    end
    $ 1242 "MoveJ"
    $ 1243 "CaptPos0" "breakAfter"
    set_tcp(p[0.0,0.0,0.0,0.0,0.0,0.0])
    movej(get_inverse_kin(CaptPos0_p, qnear=CaptPos0_q), a=0.2617993877991494, v=0.15707963267948966)
  end
  def SUB_6101():
    $ 1244 "SUB_6101" "noBreak"
    $ 1245 "ROVI_RECIPE"
    $ 1246 "If文 (not ROVI_RECIPE(GPII_WorkNo))"
    if ((not ROVI_RECIPE(read_input_integer_register(2)))):
      $ 1247 "SubPrgResult:=rovi_err"
      global SubPrgResult=rovi_err
      $ 1248 "待機: 999999.0"
      sleep(999999.0)
    end
    $ 1249 "ROVI_RESET"
    $ 1250 "If文 ( not ROVI_RESET())"
    if ((  not  ROVI_RESET())):
      $ 1251 "SubPrgResult:=rovi_err"
      global SubPrgResult=rovi_err
      $ 1252 "待機: 999999.0"
      sleep(999999.0)
    end
    $ 1253 "ROVI_CAPTURE_1"
    $ 1254 "MoveJ"
    $ 1255 "スイッチ文 CheckMST"
    switch_1 = CheckMST
    $ 1256 "ケース 0"
    if (0 == switch_1):
      $ 1257 "Master_pos" "breakAfter"
      set_tcp(p[0.0,0.09,0.42,0.0,0.0,0.0])
      movej(Master_pos, a=0.20943951023931953, v=0.10471975511965977)
    elif (1 == switch_1):
      $ 1258 "ケース 1"
      $ 1259 "Master_pos" "breakAfter"
      set_tcp(p[0.0,0.09,0.42,0.0,0.0,0.0])
      movej(Master_pos, a=0.20943951023931953, v=0.10471975511965977)
    elif (2 == switch_1):
      $ 1260 "ケース 2"
      $ 1261 "Master_posL" "breakAfter"
      set_tcp(p[0.0,0.09,0.42,0.0,0.0,0.0])
      movej(Master_posL, a=0.20943951023931953, v=0.10471975511965977)
    elif (3 == switch_1):
      $ 1262 "ケース 3"
      $ 1263 "Master_posR" "breakAfter"
      set_tcp(p[0.0,0.09,0.42,0.0,0.0,0.0])
      movej(Master_posR, a=0.20943951023931953, v=0.10471975511965977)
    end
    $ 1265 "待機: 3.0"
    sleep(3.0)
    $ 1266 "If文 ( not ROVI_CAPTURE())"
    if ((  not  ROVI_CAPTURE())):
      $ 1267 "SubPrgResult:=rovi_err"
      global SubPrgResult=rovi_err
      $ 1268 "待機: 999999.0"
      sleep(999999.0)
    end
  end
  def SUB_6102RXFF():
    $ 1438 "SUB_6102RXFF" "noBreak"
    $ 1439 "荷重の設定: k10"
    set_target_payload(0.100000, [0.135000, 0.000000, 0.225000], [10.000000, 10.000000, 10.000000, 0.000000, 0.000000, 0.000000])
    $ 1440 "UF:=ベース_const"
    global UF=p[0.0,0.0,0.0,0.0,0.0,0.0]
    $ 1441 "If文 (GPII_CheckMST>0)"
    if ((read_input_integer_register(23)>0)):
      $ 1442 "ROVI_SOLVE"
      $ 1443 "If文 (CandCnt>0)"
      if ((CandCnt>0)):
        $ 1444 "Y2:=ROVI_SOLVE()"
        global Y2=ROVI_SOLVE()
        $ 1445 "If文 (Y2[0]≟10000.)"
        if ((Y2[0] == 10000.)):
          $ 1446 "SubPrgResult:=rovi_err"
          global SubPrgResult=rovi_err
          $ 1447 "待機: 999999.0"
          sleep(999999.0)
        end
      end
      $ 1448 "UF:=Y2"
      global UF=Y2
    end
    $ 1449 "M"
    $ 1450 "MoveL"
    $ 1451 "gGD_3_M_RX" "breakAfter"
    set_tcp(p[0.0,0.09,0.42,1.894,0.0,0.0])
    movel(pose_trans(UF, gGD_3_M_RX), a=0.07, v=0.12)
    $ 1452 "待機: 1.0"
    sleep(1.0)
    $ 1453 "gGD_2_M_RX" "breakAfter"
    set_tcp(p[0.0,0.09,0.42,1.894,0.0,0.0])
    movel(pose_trans(UF, gGD_2_M_RX), a=0.07, v=0.12)
    $ 1454 "待機: 1.0"
    sleep(1.0)
    $ 1455 "設定 GPBO_BLStop=HI:Pulse 1.0"
    thread SinglePulse2252():
      write_output_boolean_register(14, True)
      sleep(1.0)
      write_output_boolean_register(14, False)
    end
    singlePulse2252 = run SinglePulse2252()
    $ 1456 "ポップアップ: ok?"
    popup("ok?", "メッセージ", False, False, blocking=True)
    $ 1457 "tm_6102_01: リセット"
    tm_6102_01 = 0
    $ 1458 "tm_6102_01: 起動"
    tm_6102_01_is_counting = True
    $ 1459 "フォース"
    sleep(0.02)
    zero_ftsensor()
    force_mode(tool_pose(), [1, 1, 1, 0, 0, 0], [0.0, 0.0, 10.0, 0.0, 0.0, 0.0], 2, [0.005, 0.005, 0.04, 0.3490658503988659, 0.3490658503988659, 0.3490658503988659])
    $ 1460 "ShakeCnt:=-1" "noBreak"
    global ShakeCnt=-1
    $ 1461 "ループ ((Currpos_p_UF0[1]>(gGD_2_M_RX[1]-HandInZ)) and (tm_6102_01<GPII_TMHandIn))" "noBreak"
    while (((Currpos_p_UF0[1]>(gGD_2_M_RX[1]-HandInZ))  and  (tm_6102_01<read_input_integer_register(12)))):
      $ 1462 "IsShake:= False " "noBreak"
      global IsShake=  False
      $ 1463 "If文 ShakeCnt<0" "noBreak"
      if (ShakeCnt<0):
        $ 1464 "NOT_SHAKE" "noBreak"
        $ 1465 "tm_6102_02: 起動" "noBreak"
        tm_6102_02_is_counting = True
        $ 1466 "待機 tm_6102_02>ShakeWaitSec" "noBreak"
        while (not(tm_6102_02>ShakeWaitSec)):
          sync()
        end
        $ 1467 "tm_6102_02: 停止" "noBreak"
        tm_6102_02_is_counting = False
        $ 1468 "tm_6102_02: リセット" "noBreak"
        tm_6102_02 = 0
        $ 1469 "ShakeCnt:=0" "noBreak"
        global ShakeCnt=0
      end
      $ 1470 "MONITOR_SPEED" "noBreak"
      $ 1471 "tm_6102_02: リセット" "noBreak"
      tm_6102_02 = 0
      $ 1472 "If文 norm(TCPSpeed[2])<TCPSpeedThZ" "noBreak"
      if (norm(TCPSpeed[2])<TCPSpeedThZ):
        $ 1473 "IsShake:= True " "noBreak"
        global IsShake=  True
        $ 1474 "If文 ShakeCnt≟0" "noBreak"
        if (ShakeCnt == 0):
          $ 1475 "tm_6102_02: 起動" "noBreak"
          tm_6102_02_is_counting = True
          $ 1476 "ループ ((tm_6102_02<1.0) and (IsShake≟ True ))" "noBreak"
          while (((tm_6102_02<1.0)  and  (IsShake ==   True  ))):
            $ 1477 "If文 norm(TCPSpeed[2])≥TCPSpeedThZ" "noBreak"
            if (norm(TCPSpeed[2]) >= TCPSpeedThZ):
              $ 1478 "IsShake:= False " "noBreak"
              global IsShake=  False
            end
          end
          $ 1479 "tm_6102_02: 停止" "noBreak"
          tm_6102_02_is_counting = False
        end
        $ 1480 "ShakeCnt:=ShakeCnt+1" "noBreak"
        global ShakeCnt=ShakeCnt+1
      end
      $ 1481 "SHAKE" "noBreak"
      $ 1482 "If文 IsShake" "noBreak"
      if (IsShake):
        $ 1483 "Sub3100_Option:=9" "noBreak"
        global Sub3100_Option=9
        $ 1484 "ループ2回" "noBreak"
        u12523u12540u12503_6 = 0
        while (u12523u12540u12503_6 < 2):
          $ 1485 "'7:RX+,8:RX-,9:RY+,10:RY-,11:RZ+,12:RZ-'" "noBreak"
          # '7:RX+,8:RX-,9:RY+,10:RY-,11:RZ+,12:RZ-'
          $ 1486 "Sub3100_Xd:=[0.,0.,0.,0.,0.,0.]" "noBreak"
          global Sub3100_Xd=[0.,0.,0.,0.,0.,0.]
          $ 1487 "Sub3100_q:=floor((Sub3100_Option-1) / 2)" "noBreak"
          global Sub3100_q=floor((Sub3100_Option-1) / 2)
          $ 1488 "Sub3100_e:=1-((Sub3100_Option-1) % 2)*2" "noBreak"
          global Sub3100_e=1-((Sub3100_Option-1) % 2)*2
          $ 1489 "Sub3100_t:=0.2" "noBreak"
          global Sub3100_t=0.2
          $ 1490 "Sub3100_Xd[Sub3100_q]=d2r(Sub3100_XdRot/2.0)*Sub3100_e" "noBreak"
          Sub3100_Xd[Sub3100_q]= d2r (Sub3100_XdRot/2.0)*Sub3100_e
          $ 1491 "speedl(Sub3100_Xd,Sub3100_aRot/2.0,Sub3100_t)" "noBreak"
          speedl(Sub3100_Xd,Sub3100_aRot/2.0,Sub3100_t)
          $ 1492 "If文 Sub3100_Option≟9" "noBreak"
          if (Sub3100_Option == 9):
            $ 1493 "Sub3100_Option:=10" "noBreak"
            global Sub3100_Option=10
          else:
            $ 1494 "Else" "noBreak"
            $ 1495 "Sub3100_Option:=9" "noBreak"
            global Sub3100_Option=9
          end
          $ 1496 "待機: 0.1" "noBreak"
          sleep(0.1)
          u12523u12540u12503_6 = u12523u12540u12503_6 + 1
        end
        $ 1497 "IsShake:= False " "noBreak"
        global IsShake=  False
      end
      $ 1498 "待機: 0.1" "noBreak"
      sleep(0.1)
    end
    end_force_mode()
    stopl(5.0)
    $ 1499 "tm_6102_01: 停止"
    tm_6102_01_is_counting = False
    $ 1500 "設定 GPBO_BLStart=HI:Pulse 1.0"
    thread SinglePulse2253():
      write_output_boolean_register(15, True)
      sleep(1.0)
      write_output_boolean_register(15, False)
    end
    singlePulse2253 = run SinglePulse2253()
    $ 1501 "待機: 1.0"
    sleep(1.0)
    $ 1502 "ポップアップ: ok?"
    popup("ok?", "メッセージ", False, False, blocking=True)
    $ 1503 "MoveL"
    $ 1504 "gGD_2_M_RX" "breakAfter"
    set_tcp(p[0.0,0.09,0.42,1.894,0.0,0.0])
    movel(pose_trans(UF, gGD_2_M_RX), a=0.07, v=0.12)
    $ 1505 "待機: 1.0"
    sleep(1.0)
    $ 1506 "gGD_3_M_RX" "breakAfter"
    set_tcp(p[0.0,0.09,0.42,1.894,0.0,0.0])
    movel(pose_trans(UF, gGD_3_M_RX), a=0.07, v=0.12)
    $ 1507 "待機: 1.0"
    sleep(1.0)
    $ 1508 "LM"
    $ 1509 "MoveL"
    $ 1510 "gGD_3_LM_RX" "breakAfter"
    set_tcp(p[0.0,0.09,0.42,1.894,0.0,0.0])
    movel(pose_trans(UF, gGD_3_LM_RX), a=0.07, v=0.12)
    $ 1511 "待機: 1.0"
    sleep(1.0)
    $ 1512 "gGD_2_LM_RX" "breakAfter"
    set_tcp(p[0.0,0.09,0.42,1.894,0.0,0.0])
    movel(pose_trans(UF, gGD_2_LM_RX), a=0.07, v=0.12)
    $ 1513 "待機: 1.0"
    sleep(1.0)
    $ 1514 "設定 GPBO_BLStop=HI:Pulse 1.0"
    thread SinglePulse2254():
      write_output_boolean_register(14, True)
      sleep(1.0)
      write_output_boolean_register(14, False)
    end
    singlePulse2254 = run SinglePulse2254()
    $ 1515 "ポップアップ: ok?"
    popup("ok?", "メッセージ", False, False, blocking=True)
    $ 1516 "tm_6102_01: リセット"
    tm_6102_01 = 0
    $ 1517 "tm_6102_01: 起動"
    tm_6102_01_is_counting = True
    $ 1518 "フォース"
    sleep(0.02)
    zero_ftsensor()
    force_mode(tool_pose(), [1, 1, 1, 0, 0, 0], [0.0, 0.0, 10.0, 0.0, 0.0, 0.0], 2, [0.005, 0.005, 0.04, 0.3490658503988659, 0.3490658503988659, 0.3490658503988659])
    $ 1519 "待機 ((Currpos_p_UF0[1]≤(gGD_2_LM_RX[1]-HandInZ)) or (tm_6102_01>GPII_TMHandIn))" "noBreak"
    while (not(((Currpos_p_UF0[1] <= (gGD_2_LM_RX[1]-HandInZ))  or  (tm_6102_01>read_input_integer_register(12))))):
      sync()
    end
    end_force_mode()
    stopl(5.0)
    $ 1520 "tm_6102_01: 停止"
    tm_6102_01_is_counting = False
    $ 1521 "設定 GPBO_BLStart=HI:Pulse 1.0"
    thread SinglePulse2255():
      write_output_boolean_register(15, True)
      sleep(1.0)
      write_output_boolean_register(15, False)
    end
    singlePulse2255 = run SinglePulse2255()
    $ 1522 "待機: 1.0"
    sleep(1.0)
    $ 1523 "ポップアップ: ok?"
    popup("ok?", "メッセージ", False, False, blocking=True)
    $ 1524 "MoveL"
    $ 1525 "gGD_2_LM_RX" "breakAfter"
    set_tcp(p[0.0,0.09,0.42,1.894,0.0,0.0])
    movel(pose_trans(UF, gGD_2_LM_RX), a=0.07, v=0.12)
    $ 1526 "待機: 1.0"
    sleep(1.0)
    $ 1527 "gGD_3_LM_RX" "breakAfter"
    set_tcp(p[0.0,0.09,0.42,1.894,0.0,0.0])
    movel(pose_trans(UF, gGD_3_LM_RX), a=0.07, v=0.12)
    $ 1528 "待機: 1.0"
    sleep(1.0)
    $ 1529 "RM"
    $ 1530 "MoveL"
    $ 1531 "gGD_3_RM_RX" "breakAfter"
    set_tcp(p[0.0,0.09,0.42,1.894,0.0,0.0])
    movel(pose_trans(UF, gGD_3_RM_RX), a=0.07, v=0.12)
    $ 1532 "待機: 1.0"
    sleep(1.0)
    $ 1533 "gGD_2_RM_RX" "breakAfter"
    set_tcp(p[0.0,0.09,0.42,1.894,0.0,0.0])
    movel(pose_trans(UF, gGD_2_RM_RX), a=0.07, v=0.12)
    $ 1534 "待機: 1.0"
    sleep(1.0)
    $ 1535 "設定 GPBO_BLStop=HI:Pulse 1.0"
    thread SinglePulse2256():
      write_output_boolean_register(14, True)
      sleep(1.0)
      write_output_boolean_register(14, False)
    end
    singlePulse2256 = run SinglePulse2256()
    $ 1536 "ポップアップ: ok?"
    popup("ok?", "メッセージ", False, False, blocking=True)
    $ 1537 "tm_6102_01: リセット"
    tm_6102_01 = 0
    $ 1538 "tm_6102_01: 起動"
    tm_6102_01_is_counting = True
    $ 1539 "フォース"
    sleep(0.02)
    zero_ftsensor()
    force_mode(tool_pose(), [1, 1, 1, 0, 0, 0], [0.0, 0.0, 10.0, 0.0, 0.0, 0.0], 2, [0.005, 0.005, 0.04, 0.3490658503988659, 0.3490658503988659, 0.3490658503988659])
    $ 1540 "待機 ((Currpos_p_UF0[1]≤(gGD_2_RM_RX[1]-HandInZ)) or (tm_6102_01>GPII_TMHandIn))" "noBreak"
    while (not(((Currpos_p_UF0[1] <= (gGD_2_RM_RX[1]-HandInZ))  or  (tm_6102_01>read_input_integer_register(12))))):
      sync()
    end
    end_force_mode()
    stopl(5.0)
    $ 1541 "tm_6102_01: 停止"
    tm_6102_01_is_counting = False
    $ 1542 "設定 GPBO_BLStart=HI:Pulse 1.0"
    thread SinglePulse2257():
      write_output_boolean_register(15, True)
      sleep(1.0)
      write_output_boolean_register(15, False)
    end
    singlePulse2257 = run SinglePulse2257()
    $ 1543 "待機: 1.0"
    sleep(1.0)
    $ 1544 "ポップアップ: ok?"
    popup("ok?", "メッセージ", False, False, blocking=True)
    $ 1545 "MoveL"
    $ 1546 "gGD_2_RM_RX" "breakAfter"
    set_tcp(p[0.0,0.09,0.42,1.894,0.0,0.0])
    movel(pose_trans(UF, gGD_2_RM_RX), a=0.07, v=0.12)
    $ 1547 "待機: 1.0"
    sleep(1.0)
    $ 1548 "gGD_3_RM_RX" "breakAfter"
    set_tcp(p[0.0,0.09,0.42,1.894,0.0,0.0])
    movel(pose_trans(UF, gGD_3_RM_RX), a=0.07, v=0.12)
    $ 1549 "待機: 1.0"
    sleep(1.0)
    $ 1550 "MoveL"
    $ 1551 "gHome_Position" "breakAfter"
    set_tcp(p[0.0,0.09,0.42,0.0,0.0,0.0])
    movel(gHome_Position, a=0.07, v=0.12)
  end
  def SUB_6402():
    $ 1552 "SUB_6402" "noBreak"
    $ 1553 "INITIALIZE"
    $ 1554 "荷重の設定: k10"
    set_target_payload(0.100000, [0.135000, 0.000000, 0.225000], [10.000000, 10.000000, 10.000000, 0.000000, 0.000000, 0.000000])
    $ 1555 "ROVI_RECIPE"
    $ 1556 "If文 ( not ROVI_RECIPE(GPII_ConveyorNo))"
    if ((  not  ROVI_RECIPE(read_input_integer_register(1)))):
      $ 1557 "SubPrgResult:=rovi_err"
      global SubPrgResult=rovi_err
      $ 1558 "待機: 999999.0"
      sleep(999999.0)
    end
    $ 1559 "ROVI_RESET"
    $ 1560 "If文 ( not ROVI_RESET())"
    if ((  not  ROVI_RESET())):
      $ 1561 "SubPrgResult:=rovi_err"
      global SubPrgResult=rovi_err
      $ 1562 "待機: 999999.0"
      sleep(999999.0)
    end
    $ 1563 "ROVI_CAPTURE"
    $ 1564 "MoveL"
    $ 1565 "Capt_CV_M" "breakAfter"
    set_tcp(p[0.0,0.09,0.42,0.0,0.0,0.0])
    movel(Capt_CV_M, a=0.07, v=0.2)
    $ 1566 "待機: 2.0"
    sleep(2.0)
    $ 1567 "If文 ( not ROVI_CAPTURE())"
    if ((  not  ROVI_CAPTURE())):
      $ 1568 "SubPrgResult:=rovi_err"
      global SubPrgResult=rovi_err
      $ 1569 "待機: 999999.0"
      sleep(999999.0)
    end
  end
  def SUB_7001():
    $ 1570 "SUB_7001" "noBreak"
    $ 1571 "荷重の設定: k10"
    set_target_payload(0.100000, [0.135000, 0.000000, 0.225000], [10.000000, 10.000000, 10.000000, 0.000000, 0.000000, 0.000000])
    $ 1572 "MoveL"
    $ 1573 "gTAIHI_pos1" "breakAfter"
    set_tcp(p[0.0,0.09,0.42,0.0,0.0,0.0])
    movel(gTAIHI_pos1, a=0.07, v=0.12)
    $ 1574 "gTAIHI_pos2" "breakAfter"
    set_tcp(p[0.0,0.09,0.42,0.0,0.0,0.0])
    movel(gTAIHI_pos2, a=0.07, v=0.12)
    $ 1575 "gTAIHI_pos3" "breakAfter"
    set_tcp(p[0.0,0.09,0.42,0.0,0.0,0.0])
    movel(gTAIHI_pos3, a=0.07, v=0.12)
    $ 1576 "gTAIHI_pos4" "breakAfter"
    set_tcp(p[0.0,0.09,0.42,0.0,0.0,0.0])
    movel(gTAIHI_pos4, a=0.07, v=0.12)
    $ 1577 "gTAIHI_pos5" "breakAfter"
    set_tcp(p[0.0,0.09,0.42,0.0,0.0,0.0])
    movel(gTAIHI_pos5, a=0.07, v=0.12)
  end
  def SUB_7002():
    $ 1578 "SUB_7002" "noBreak"
    $ 1579 "荷重の設定: k10"
    set_target_payload(0.100000, [0.135000, 0.000000, 0.225000], [10.000000, 10.000000, 10.000000, 0.000000, 0.000000, 0.000000])
    $ 1580 "MoveL"
    $ 1581 "gTAIHI_pos5" "breakAfter"
    movel(gTAIHI_pos5, a=0.07, v=0.12)
    $ 1582 "gTAIHI_pos4" "breakAfter"
    movel(gTAIHI_pos4, a=0.07, v=0.12)
    $ 1583 "gTAIHI_pos3" "breakAfter"
    movel(gTAIHI_pos3, a=0.07, v=0.12)
    $ 1584 "gTAIHI_pos2" "breakAfter"
    movel(gTAIHI_pos2, a=0.07, v=0.12)
    $ 1585 "gTAIHI_pos1" "breakAfter"
    movel(gTAIHI_pos1, a=0.07, v=0.12)
    $ 1586 "gHome_Position" "breakAfter"
    movel(gHome_Position, a=0.07, v=0.12)
  end
  $ 2 "開始前シーケンス"
  $ 3 "スクリプト: ROVI_RESET.script"
  def ROVI_RESET():
    if (not socket_open(host,port,socket_name)):
      rovi_err=902
      return False
    end
    socket_send_line("X0()",socket_name)
    ret=socket_read_line(socket_name,socket_timeout)
    if (ret == "OK"):
      rovi_err=0
    elif (ret == "NG"):
      rovi_err=to_num(socket_read_line(socket_name,socket_timeout))
    else:
      ret="NG"
      rovi_err=903
    end
    socket_close(socket_name)
    if (rovi_err != 0):
      if (is_popup):
        popup(str_cat(ret,rovi_err),title="X0",warning=True,blocking=True)
      end
      return False
    else:
      return True
    end
  end
  $ 4 "スクリプト: ROVI_CAPTURE.script"
  def ROVI_CAPTURE():
    Y1=[0.0,0.0,0.0,0.0]
  #  p=get_actual_tool_flange_pose()
    p=Bucket
    if (not socket_open(host,port,socket_name)):
      rovi_err=902
      return False
    end
    socket_send_string("X1(",socket_name)
    socket_send_string(p[0],socket_name)
    socket_send_string(",",socket_name)
    socket_send_string(p[1],socket_name)
    socket_send_string(",",socket_name)
    socket_send_string(p[2],socket_name)
    socket_send_string(",",socket_name)
    socket_send_string(p[3],socket_name)
    socket_send_string(",",socket_name)
    socket_send_string(p[4],socket_name)
    socket_send_string(",",socket_name)
    socket_send_string(p[5],socket_name)
    socket_send_line(")",socket_name)
    ret=socket_read_line(socket_name,socket_timeout)
    if (ret == "OK"):
      rovi_err=0
      f=socket_read_ascii_float(4,socket_name,socket_timeout)
      while (f[0]!=4):
        sleep(0.3)
        f=socket_read_ascii_float(4,socket_name,socket_timeout)
      end
      i=0
      while (i<4):
        Y1[i]=f[i+1]
        i=i+1
      end
    elif (ret == "NG"):
      rovi_err=to_num(socket_read_line(socket_name,socket_timeout))
    else:
      ret="NG"
      rovi_err=903
    end
    socket_close(socket_name)
    if (rovi_err != 0):
      if (is_popup):
        popup(str_cat(ret,rovi_err),title="X1",warning=True,blocking=True)
      end
      return False
    else:
      return True
    end
  end
  $ 5 "スクリプト: ROVI_SOLVE.script"
  def ROVI_SOLVE(is_popup=is_popup):
    buf=p[10000.0,0.0,0.0,0.0,0.0,0.0]
    if (not socket_open(host,port,socket_name)):
      rovi_err=902
      return False
    end
    socket_send_line("X2()",socket_name)
    ret=socket_read_line(socket_name,socket_timeout)
    if (ret == "OK"):
      rovi_err=0
      f=socket_read_ascii_float(6,socket_name,socket_timeout)
      while (f[0]!=6):
        sleep(0.3)
        f=socket_read_ascii_float(6,socket_name,socket_timeout)
      end
      counter=0
      while (counter<6):
        buf[counter]=f[counter+1]
        counter=counter+1
      end
    elif (ret == "NG"):
      rovi_err=to_num(socket_read_line(socket_name,socket_timeout))
    else:
      ret="NG"
      rovi_err=903
    end
    sleep(1.0)
    socket_close(socket_name)
    if (rovi_err != 0):
      if (is_popup):
        popup(str_cat(ret,rovi_err),title="X2",warning=True,blocking=True)
      end
    end
    return buf
  end
  $ 6 "スクリプト: ROVI_RECIPE.script"
  def ROVI_RECIPE(recipe):
    if (not socket_open(host,port,socket_name)):
      rovi_err=902
      return False
    end
    socket_send_line(str_cat(str_cat("X3(",recipe),")"),socket_name)
    ret=socket_read_line(socket_name,socket_timeout)
    if (ret == "OK"):
      rovi_err=0
    elif (ret == "NG"):
      rovi_err=to_num(socket_read_line(socket_name,socket_timeout))
    else:
      ret="NG"
      rovi_err=903
    end
    socket_close(socket_name)
    if (rovi_err != 0):
      if (is_popup):
        popup(str_cat(ret,rovi_err),title="X3",warning=True,blocking=True)
      end
      return False
    else:
      return True
    end
  end
  $ 7 "スクリプト: ROVI_PARAM.script"
  def ROVI_PARAM(prm_name,prm_value=None):
    Y8=0.0
    if (not socket_open(host,port,socket_name)):
      rovi_err=902
      return False
    end
    socket_send_string("X8(",socket_name)
    socket_send_string(prm_name,socket_name)
    if (prm_value != None):
      socket_send_string(" ",socket_name)
      socket_send_string(prm_value,socket_name)
    end
    socket_send_line(")",socket_name)
    ret=socket_read_line(socket_name,socket_timeout)
    if (ret == "OK"):
      rovi_err=0
      if (prm_value == None):  # rosparam get
        Y8=to_num(socket_read_line(socket_name,socket_timeout))
      else:    # rosparam set
        f=1
      end
    elif (ret == "NG"):
      rovi_err=to_num(socket_read_line(socket_name,socket_timeout))
    else:
      ret="NG"
      rovi_err=903
    end
    socket_close(socket_name)
    if (rovi_err != 0):
      if (is_popup):
        popup(str_cat(ret,rovi_err),title="X8",warning=True,blocking=True)
      end
      return False
    else:
      return True
    end
  end
  $ 8 "スクリプト: STATUS_CONTROL.script"
  def CHECK_VT_STATUS():
    write_output_boolean_register(8, read_input_boolean_register(64))   # GPBO_PCOK
    write_output_boolean_register(9, read_input_boolean_register(65))   # GPBO_YCAMOK
    write_output_integer_register(5, read_input_integer_register(24))   # GPIO_PayloadNo
  end
  $ 9 "スクリプト: CYCLE_CONTROL.script"
  def GET_REG(prg_no):
    WorkPosNo=read_input_integer_register(4)-1                       # GPII_WorkPosNo
    CaptIndex[WorkPosNo]=read_input_integer_register(21)-1           # GPII_CaptColNo
    CaptRowNo=read_input_integer_register(20)-1        # GPII_CaptRowNo
    CaptStepZ=read_input_integer_register(6) / 1000.0         # GPII_CaptStepZ
    ReCaptNo=0
    if (prg_no==1203):
      ReCaptNo=read_input_integer_register(22)                # GPII_ReCaptNo
    end
    ReCaptZ=read_input_integer_register(7) / 1000.0         # GPII_ReCaptZ
    CutOffZDef=read_input_integer_register(11) / 1000.0          # GPII_CutOffZ
    CrankDepthFull=read_input_integer_register(10) / 1000.0   # GPII_FullDepth
  end

  def POSE_SUB(p, teach_frame):
    return pose_trans(inv(teach_frame), p)
  end

  def GET_BUCKET_UPPER(pos=0):
    if UseNewCaptPos:
      p=POSE_SUB(CaptPoint_C, BucketM)
      pX=[BKWidth/2,CaptPointL_dX,BKWidth-CaptPointR_dX]
      p[0]=pX[pos]
    else:
      captpos=[CaptPoint_C,CaptPoint_L,CaptPoint_R]
      p=captpos[pos]
      p=POSE_SUB(p, BucketM)
    end
    return p
  end

  def SET_BUCKET_DEF():
    BucketM=pBucketM
    if (WorkPosNo<0):
      Bucket=pBucketC
    else:
      Bucket=pBucket[WorkPosNo]
    end
  end

  def SET_BUCKET():
    SET_BUCKET_DEF()
    Bucket[2]=Bucket[2]-CaptStepZ*CaptRowNo
  end

  def SET_CV():
    CV=pCV
  end

  def SET_CAPT_INDEX():
    CaptIndexWk=CaptIndex[WorkPosNo]
    ReCaptZWk=0
    if (prg_no==1203):
      if   (ReCaptNo==0):
        if (CaptIndexWk==0):
          if (0<=DistPillarBak):
            CaptIndexWk=1
          else:
            CaptIndexWk=2
          end
          ReCaptZWk=0
        else:
          CaptIndexWk=0
          ReCaptZWk=0
        end
      elif (ReCaptNo==1):
        if (CaptIndexWk==0):
          CaptIndexWk=0
          ReCaptZWk=-ReCaptZ
        else:
          CaptIndexWk=CaptIndexWk
          ReCaptZWk=-ReCaptZ
        end
      else:
        if (CaptIndexWk==0):
          CaptIndexWk=0
          ReCaptZWk=ReCaptZ
        else:
          CaptIndexWk=CaptIndexWk
          ReCaptZWk=ReCaptZ
        end
      end
    end
  end

  def GET_CAPTPOS():
    SET_BUCKET()
    SET_CAPT_INDEX()
    if UseNewCaptPos:
      p=GET_BUCKET_UPPER(CaptIndexWk)
      p[2]=p[2]-ReCaptZWk
    else:
      captpos=[CaptPoint_C,CaptPoint_L,CaptPoint_R]
      p=captpos[CaptIndexWk]
      p[2]=p[2]-ReCaptZWk
      p=POSE_SUB(p, BucketM)
    end
    return p
  end

  def CHECK_CAPTPOS():
    isOK=((CaptStepZ*(read_input_integer_register(20)-1)) < (read_input_integer_register(9) / 1000.0))
    return isOK
  end

  def GET_ZSLIDE_POS(p):
    p[2]=p[2]-CaptStepZ*CaptRowNo
    return p
  end

  def END_CYCLE():
    stopl(1.2)
    end_force_mode()
    end_freedrive_mode()
    socket_close(socket_name)
  end

  def CHECK_SPEED(smax,f=[1,1,1,1,1,1]):
    s=TCPSpeed
    i=0
    while (i<6):
      if ((f[i]==1) and (smax[i]<s[i])):
        return False
      end
      i=i+1
    end
    return True
  end
  $ 10 "スクリプト: ZONE_CONTROL.script"
  def GET_DIST(P1, P2):
    return pose_dist(P1, P2)
  end
  def CHECK_DIST_NEAR(P1, P2, th):
    return (GET_DIST(P1, P2) < th)
  end
  def DIST_HOME():
    return pose_dist(gHome_Position,CurrPos_p)
  end

  def CHECK_HOME():
    return (DIST_HOME()<ZoneDistTh)
  end

  def DIST_CVUpper():
    if (read_input_integer_register(4)==1):
      p=g2GD_pos1
    else:
      p=g1GD_pos1
    end
    return pose_dist(p,CurrPos_p)
  end

  def CHECK_CVUpper():
    return (DIST_CVUpper()<ZoneDistTh)
  end

  def CHECK_RB_POS(prg_no):
    ret=True
    if (prg_no==1001):
      ret=CHECK_EVAC()
    end
    if ((prg_no==1201) or (prg_no==1401) or (prg_no==1402) or (prg_no==6001) or (prg_no==6101) or (prg_no==6401) or (prg_no==6102) or (prg_no==7001)):
      ret=CHECK_HOME()
    end
    if ((prg_no==1002) or (prg_no==1241) or (prg_no==1261)):
      ret=CHECK_BKInside()
    end
    if (prg_no==1251):
      ret=(CHECK_HOME() or CHECK_CVUpper())
    end
    if (ret != True):
      SubPrgResult=801
      sleep(999999.0)
    end
  end

  def DIST_ORIGIN():
    p=CurrPos_p
    o=p
    o[0]=0.0
    o[1]=0.0
    return pose_dist(o,p)
  end

  def CHECK_EVAC_ORG():
    return (EvacRadiusTh<DIST_ORIGIN())
  end

  def CHECK_EVAC_X():
    return (EvacXTh[0]<CurrPos_p[0] and CurrPos_p[0]<EvacXTh[1])
  end

  def CHECK_EVAC_Y():
    return (EvacYTh[0]<CurrPos_p[1] and CurrPos_p[1]<EvacYTh[1])
  end

  def CHECK_EVAC_Z():
    return (EvacZTh[0]<CurrPos_p[2])
  end

  def CHECK_EVAC():
    ret=True
    ret=(ret and CHECK_EVAC_ORG())
    ret=(ret and CHECK_EVAC_X())
    ret=(ret and CHECK_EVAC_Y())
    ret=(ret and CHECK_EVAC_Z())
    return ret
  end

  def CHECK_BKInside():
    ret=True
    pos=read_input_integer_register(4)
    if (pos>2):
      ret=False
    else:
      if (not read_input_boolean_register(13+pos)):
        ret=False
        ver_3=read_input_boolean_register(13+pos)
      else:
        bk=pBucket[pos-1]
        if (pos==1):
          ret=(ret and CurrPos_p[0]>ZoneHomeX)
          ret=(ret and bk[1]-(BucketWidth-ZoneBucketGap)<CurrPos_p[1] and CurrPos_p[1]<bk[1]-ZoneBucketGap)
        elif (pos==2):
          ret=(ret and CurrPos_p[0]<-ZoneHomeX)
          ret=(ret and bk[1]+ZoneBucketGap<CurrPos_p[1] and CurrPos_p[1]<bk[1]+(BucketWidth-ZoneBucketGap))
        end
      end
    end
    return ret
  end

  def CHECK_CVOutside():
    ret=True
    ret=(ret and gCV_11_M[0]-Zone6ThX<CurrPos_p[0])
    ret=(ret and CurrPos_p[0]<gCV_11_M[0]+Zone6ThX)
    ret=(ret and gCV_11_M[1]-Zone6ThY<CurrPos_p[1])
    ret=(ret and CurrPos_p[1]<gCV_11_M[1]+Zone6ThY)
    return (not ret)
  end

  def CHECK_ZONE(no):
    if (no==1):
      return (CurrPos_p[2]>=Zone1ZTh)
    elif (no==2):
      return (CurrPos_p[0]>ZoneHomeX)
    elif (no==3):
      return (CurrPos_p[0]<-ZoneHomeX)
    elif (no==4):
      return CHECK_CVUpper()
    elif (no==5):
      return CHECK_BKInside()
    elif (no==6):
      return CHECK_CVOutside()
    end
  end
  $ 11 "スクリプト: ALIGN_AXIS.script"
  def GET_NORM_VEC(p,axis=2):
    rot=p[0.0, 0.0, 0.0, p[3], p[4], p[5]]
    vec=p[0.0, 0.0, 0.0, 0.0, 0.0, 0.0]
    vec[axis]=1.0
    norm_p=pose_trans(rot,vec)
    return [norm_p[0], norm_p[1], norm_p[2]]
  end

  def GET_INNER_PRODUCT(v1,v2):
    return v1[0]*v2[0]+v1[1]*v2[1]+v1[2]*v2[2]
  end
  def GET_OUTER_PRODUCT(v1,v2):
    x=v1[1]*v2[2]-v1[2]*v2[1]
    y=v1[2]*v2[0]-v1[0]*v2[2]
    z=v1[0]*v2[1]-v1[1]*v2[0]
    return [x,y,z]
  end
  def GET_THETA(v1,v2):
  #  cos=GET_INNER_PRODUCT(v1,v2) / norm(v1) / norm(v2)
    cos=GET_INNER_PRODUCT(v1,v2)
    g_cos=cos
    theta=norm(acos(cos))
    return theta
  end

  def GET_ALIGNED_POSE(target,feature,axis=2):
    feature_from_target=pose_trans(pose_inv(target),feature)
    g_f_from_t=feature_from_target
    nz_feature_from_target=GET_NORM_VEC(feature_from_target,axis)
    g_nz_f_from_t=nz_feature_from_target
    nz_target_from_target=[0.0, 0.0, 0.0]
    nz_target_from_target[axis]=1.0
    g_nz_t_from_t=nz_target_from_target

    theta=GET_THETA(nz_feature_from_target,nz_target_from_target)
    g_theta=theta
    rot_vec_n=normalize(GET_OUTER_PRODUCT(nz_target_from_target,nz_feature_from_target))

    if theta>d2r(90.0):
      theta=theta-d2r(180.0)
    end
    rot_vec=rot_vec_n * (theta)
    rot_p=p[0.0,0.0,0.0,rot_vec[0],rot_vec[1],rot_vec[2]]
    return pose_trans(target,rot_p)
  end
  def GET_ALIGNED_TCP(feature,axis=2):
    tcp=get_actual_tcp_pose()
    return GET_ALIGNED_POSE(tcp,feature,axis)
  end

  $ 12 "スクリプト: ROTATE_CONTROL.script"
  def GET_TCP_FORCE_TOOL():
    force_torque=get_tcp_force()
    force_B=p[force_torque[0], force_torque[1], force_torque[2], 0, 0, 0]
    torque_B=p[force_torque[3], force_torque[4], force_torque[5], 0, 0, 0]
    tcp=get_actual_tcp_pose()
    rotation_BT=p[0, 0, 0, tcp[3], tcp[4], tcp[5]]
    force_T=pose_trans(pose_inv(rotation_BT), force_B)
    torque_T=pose_trans(pose_inv(rotation_BT), torque_B)
    force_torque_T=p[force_T[0], force_T[1], force_T[2], torque_T[0], torque_T[1], torque_T[2]]
    return force_torque_T
  end

  def CHECK_VALUE_RZ():
    return True
  end

  def GET_FORCE_VALUE_RZ(target):
    PoseSub= pose_sub (CurrPos_p,target)
    RYSub=r2d(PoseSub[4])
    RZSub=r2d(PoseSub[5])
  #  if (RYSub<RZSupRYRange[0] or RZSupRYRange[1]<RYSub):
  #    RZSupForceVal=0.0
  #    return RZSupForceVal
  #  end
    if (RZSub<0):
      RZMin=RZSupDegMin[0]
      RZRatio=RZSupRatio[0]
      RZOffset=RZSupOffset[0]
    else:
      RZMin=RZSupDegMin[1]
      RZRatio=RZSupRatio[1]
      RZOffset=-RZSupOffset[1]
    end
    if (norm(RZSub) >= norm(RZMin)):
      RZSupForceVal=(RZMin-RZSub)*RZRatio+RZOffset
    else:
      RZSupForceVal=0
    end
    if (RZSupForceVal<RZSupForceRange[0]):
      RZSupForceVal=RZSupForceRange[0]
    elif (RZSupForceRange[1]<RZSupForceVal):
      RZSupForceVal=RZSupForceRange[1]
    end
    if (RYSub<RZSupRYRange[0] or RZSupRYRange[1]<RYSub):
      RZSupForceVal=0
    end
    if ((not UseRZSupStep1) and (ForceStep==1)):
      RZSupForceVal=0
    end
    return RZSupForceVal
  end

  def GET_CVCORR_RZ(target):
    PoseSub=pose_sub(CurrPos_p,target)
    RYSub=r2d(PoseSub[4])
    if (RYSub<0):
      RYMin=-CVCorrDegMin[0]
      RZRatio=CVCorrRatio[0]
      RZOffset=-CVCorrOffset[0]
    else:
      RYMin=-CVCorrDegMin[1]
      RZRatio=CVCorrRatio[1]
      RZOffset=CVCorrOffset[1]
    end
    if (norm(RYSub) >= norm(RYMin)):
      CVCorrRZVal=RYSub*RZRatio+RZOffset
    else:
      CVCorrRZVal=0
    end
    return CVCorrRZVal
  end
  $ 209 "u12473u12524u12483u12489_2"
  thread u12473u12524u12483u12489_2():
    while (True):
      $ 210 "Sub3100_GPII18:=GPII_RunOption"
      global Sub3100_GPII18=read_input_integer_register(18)
      $ 211 "CurrPos=get_actual_tool_flange_pose()"
      CurrPos=get_actual_tool_flange_pose()
      $ 212 "CurrPos_p=get_actual_tcp_pose()"
      CurrPos_p= get_actual_tcp_pose ()
      $ 213 "Currpos_p_UF0=pose_trans(pose_inv(UF), CurrPos_p)"
      Currpos_p_UF0= pose_trans ( pose_inv (UF), CurrPos_p)
      $ 214 "TCPSpeed:=get_actual_tcp_speed()"
      global TCPSpeed=get_actual_tcp_speed()
      $ 215 "TCPForce:=get_tcp_force()"
      global TCPForce=get_tcp_force()
      $ 216 "設定 GPBO_RBHome=CHECK_HOME()"
      write_output_boolean_register(12, CHECK_HOME())
      $ 217 "設定 GPBO_AllowGoHom=CHECK_EVAC()"
      write_output_boolean_register(16, CHECK_EVAC())
      $ 218 "設定 GPBO_Zone01=CHECK_ZONE(1)"
      write_output_boolean_register(24, CHECK_ZONE(1))
      $ 219 "設定 GPBO_Zone02=CHECK_ZONE(2)"
      write_output_boolean_register(25, CHECK_ZONE(2))
      $ 220 "設定 GPBO_Zone03=CHECK_ZONE(3)"
      write_output_boolean_register(26, CHECK_ZONE(3))
      $ 221 "設定 GPBO_Zone04=CHECK_ZONE(4)"
      write_output_boolean_register(27, CHECK_ZONE(4))
      $ 222 "設定 GPBO_Zone05=CHECK_ZONE(5)"
      write_output_boolean_register(28, CHECK_ZONE(5))
      $ 223 "設定 GPBO_Zone06=CHECK_ZONE(6)"
      write_output_boolean_register(29, CHECK_ZONE(6))
      $ 224 "CHECK_VT_STATUS()"
      CHECK_VT_STATUS()
      $ 225 "sync()"
      sync()
    end
  end
  threadId_u12473u12524u12483u12489_2 = run u12473u12524u12483u12489_2()
  while (True):
    $ 14 "ロボットプログラム"
    $ 15 "position_deviation_warning(True,0.4)"
    position_deviation_warning(True,0.4)
    $ 16 "荷重の設定: k10"
    set_target_payload(0.100000, [0.135000, 0.000000, 0.225000], [10.000000, 10.000000, 10.000000, 0.000000, 0.000000, 0.000000])
    $ 17 "設定"
    set_tcp(p[0.0,0.09,0.42,0.0,0.0,0.0])
    $ 18 "CutOffTCP:=get_tcp_offset()"
    global CutOffTCP=get_tcp_offset()
    $ 19 "設定 GPIO_PrgNo=0"
    write_output_integer_register(0, 0)
    $ 20 "設定 GPBO_PrgBegin=オフ"
    write_output_boolean_register(4, False)
    $ 21 "設定 GPBO_PrgEnd=オフ"
    write_output_boolean_register(5, False)
    $ 22 "設定 GPBO_PrgRun=オフ"
    write_output_boolean_register(6, False)
    $ 23 "設定 GPBO_BKPosDone=オフ"
    write_output_boolean_register(13, False)
    $ 24 "設定 GPBO_BLStop=オフ"
    write_output_boolean_register(14, False)
    $ 25 "設定 GPBO_BLStart=オフ"
    write_output_boolean_register(15, False)
    $ 26 "設定 GPBO_Released=オフ"
    write_output_boolean_register(17, False)
    $ 27 "待機 GPBI_PrgStart=LO"
    while (read_input_boolean_register(4) == True):
      sync()
    end
    $ 28 "待機 GPBI_PrgStart=HI"
    while (read_input_boolean_register(4) == False):
      sync()
    end
    $ 29 "設定 GPIO_PrgResult=0"
    write_output_integer_register(1, 0)
    $ 30 "prg_no:=GPII_PrgNo"
    global prg_no=read_input_integer_register(0)
    $ 31 "If文 ( not GPBI_PrgStop≠ False )"
    global thread_flag_31=0
    thread Thread_if_31():
      $ 32 "CHECK_RB_POS(prg_no)"
      CHECK_RB_POS(prg_no)
      $ 33 "設定 GPIO_PrgNo=prg_no"
      write_output_integer_register(0, prg_no)
      $ 34 "待機: 0.1"
      sleep(0.1)
      $ 35 "設定 GPBO_PrgBegin=HI:Pulse 1.0"
      thread SinglePulse2258():
        write_output_boolean_register(4, True)
        sleep(1.0)
        write_output_boolean_register(4, False)
      end
      singlePulse2258 = run SinglePulse2258()
      $ 36 "SubPrgResult:=100"
      global SubPrgResult=100
      $ 37 "If文 (SubPrgResult≟100)"
      global thread_flag_37=0
      thread Thread_if_37():
        $ 38 "GET_REG(prg_no)"
        GET_REG(prg_no)
        $ 39 "スイッチ文 prg_no"
        switch_1 = prg_no
        $ 40 "ケース 1001"
        if (1001 == switch_1):
          $ 41 "CHECK_RB_POS(prg_no)"
          CHECK_RB_POS(prg_no)
          $ 42 "設定 GPIO_SubPrgNo=001"
          write_output_integer_register(2, 001)
          $ 43 "呼び出し SUB_001"
          SUB_001()
        elif (1002 == switch_1):
          $ 44 "ケース 1002"
          $ 45 "設定 GPIO_SubPrgNo=102"
          write_output_integer_register(2, 102)
          $ 46 "呼び出し SUB_002"
          SUB_002()
          $ 47 "設定 GPIO_SubPrgNo=001"
          write_output_integer_register(2, 001)
          $ 48 "呼び出し SUB_001"
          SUB_001()
        elif (1201 == switch_1):
          $ 49 "ケース 1201"
          $ 50 "設定 GPIO_SubPrgNo=101"
          write_output_integer_register(2, 101)
          $ 51 "呼び出し SUB_101"
          SUB_101()
          $ 52 "設定 GPIO_SubPrgNo=102"
          write_output_integer_register(2, 102)
          $ 53 "呼び出し SUB_102"
          SUB_102()
          $ 54 "設定 GPIO_SubPrgNo=104"
          write_output_integer_register(2, 104)
          $ 58 "呼び出し SUB_104RXFF"
          SUB_104RXFF()
          $ 59 "設定 GPIO_SubPrgNo=105"
          write_output_integer_register(2, 105)
          $ 60 "呼び出し SUB_105"
          SUB_105()
          $ 61 "設定 GPIO_SubPrgNo=106"
          write_output_integer_register(2, 106)
          $ 62 "呼び出し SUB_106"
          SUB_106()
          $ 63 "設定 GPIO_SubPrgNo=121"
          write_output_integer_register(2, 121)
          $ 64 "呼び出し SUB_121"
          SUB_121()
          $ 65 "設定 GPIO_SubPrgNo=122"
          write_output_integer_register(2, 122)
          $ 66 "呼び出し SUB_122"
          SUB_122()
          $ 67 "設定 GPIO_SubPrgNo=001"
          write_output_integer_register(2, 001)
          $ 68 "呼び出し SUB_001"
          SUB_001()
          $ 69 "If文 (CandCnt≟1)"
          if ((CandCnt == 1)):
            $ 70 "SubPrgResult:=990"
            global SubPrgResult=990
            $ 71 "待機: 999999.0"
            sleep(999999.0)
          end
        elif (1202 == switch_1):
          $ 72 "ケース 1202"
          $ 73 "設定 GPIO_SubPrgNo=102"
          write_output_integer_register(2, 102)
          $ 74 "呼び出し SUB_102"
          SUB_102()
          $ 75 "設定 GPIO_SubPrgNo=104"
          write_output_integer_register(2, 104)
          $ 80 "呼び出し SUB_104RXFF"
          SUB_104RXFF()
          $ 81 "設定 GPIO_SubPrgNo=105"
          write_output_integer_register(2, 105)
          $ 82 "呼び出し SUB_105"
          SUB_105()
          $ 83 "設定 GPIO_SubPrgNo=106"
          write_output_integer_register(2, 106)
          $ 84 "呼び出し SUB_106"
          SUB_106()
          $ 85 "設定 GPIO_SubPrgNo=121"
          write_output_integer_register(2, 121)
          $ 86 "呼び出し SUB_121"
          SUB_121()
          $ 87 "設定 GPIO_SubPrgNo=122"
          write_output_integer_register(2, 122)
          $ 88 "呼び出し SUB_122"
          SUB_122()
          $ 89 "設定 GPIO_SubPrgNo=001"
          write_output_integer_register(2, 001)
          $ 90 "呼び出し SUB_001"
          SUB_001()
          $ 91 "If文 (CandCnt≟1)"
          if ((CandCnt == 1)):
            $ 92 "SubPrgResult:=990"
            global SubPrgResult=990
            $ 93 "待機: 999999.0"
            sleep(999999.0)
          end
        elif (1203 == switch_1):
          $ 94 "ケース 1203"
          $ 95 "設定 GPIO_SubPrgNo=103"
          write_output_integer_register(2, 103)
          $ 96 "呼び出し SUB_103"
          SUB_103()
          $ 97 "設定 GPIO_SubPrgNo=104"
          write_output_integer_register(2, 104)
          $ 101 "呼び出し SUB_104RXFF"
          SUB_104RXFF()
          $ 102 "設定 GPIO_SubPrgNo=105"
          write_output_integer_register(2, 105)
          $ 103 "呼び出し SUB_105"
          SUB_105()
          $ 104 "設定 GPIO_SubPrgNo=106"
          write_output_integer_register(2, 106)
          $ 105 "呼び出し SUB_106"
          SUB_106()
          $ 106 "設定 GPIO_SubPrgNo=121"
          write_output_integer_register(2, 121)
          $ 107 "呼び出し SUB_121"
          SUB_121()
          $ 108 "設定 GPIO_SubPrgNo=122"
          write_output_integer_register(2, 122)
          $ 109 "呼び出し SUB_122"
          SUB_122()
          $ 110 "設定 GPIO_SubPrgNo=001"
          write_output_integer_register(2, 001)
          $ 111 "呼び出し SUB_001"
          SUB_001()
          $ 112 "If文 (CandCnt≟1)"
          if ((CandCnt == 1)):
            $ 113 "SubPrgResult:=990"
            global SubPrgResult=990
            $ 114 "待機: 999999.0"
            sleep(999999.0)
          end
        elif (1241 == switch_1):
          $ 115 "ケース 1241"
          $ 116 "設定 GPIO_SubPrgNo=106"
          write_output_integer_register(2, 106)
          $ 117 "呼び出し SUB_106"
          SUB_106()
          $ 118 "設定 GPIO_SubPrgNo=121"
          write_output_integer_register(2, 121)
          $ 119 "呼び出し SUB_121"
          SUB_121()
          $ 120 "設定 GPIO_SubPrgNo=122"
          write_output_integer_register(2, 122)
          $ 121 "呼び出し SUB_122"
          SUB_122()
          $ 122 "設定 GPIO_SubPrgNo=001"
          write_output_integer_register(2, 001)
          $ 123 "呼び出し SUB_001"
          SUB_001()
        elif (1251 == switch_1):
          $ 124 "ケース 1251"
          $ 125 "設定 GPIO_SubPrgNo=120"
          write_output_integer_register(2, 120)
          $ 126 "呼び出し SUB_120"
          SUB_120()
          $ 127 "設定 GPIO_SubPrgNo=121"
          write_output_integer_register(2, 121)
          $ 128 "呼び出し SUB_121"
          SUB_121()
          $ 129 "設定 GPIO_SubPrgNo=122"
          write_output_integer_register(2, 122)
          $ 130 "呼び出し SUB_122"
          SUB_122()
          $ 131 "設定 GPIO_SubPrgNo=001"
          write_output_integer_register(2, 001)
          $ 132 "呼び出し SUB_001"
          SUB_001()
        elif (1261 == switch_1):
          $ 133 "ケース 1261"
          $ 134 "設定 GPIO_SubPrgNo=161"
          write_output_integer_register(2, 161)
          $ 135 "呼び出し SUB_161"
          SUB_161()
          $ 136 "設定 GPIO_SubPrgNo=001"
          write_output_integer_register(2, 001)
          $ 137 "呼び出し SUB_001"
          SUB_001()
        elif (1281 == switch_1):
          $ 138 "ケース 1281"
          $ 139 "設定 GPIO_SubPrgNo=181"
          write_output_integer_register(2, 181)
          $ 140 "呼び出し SUB_181"
          SUB_181()
          $ 141 "設定 GPIO_SubPrgNo=001"
          write_output_integer_register(2, 001)
          $ 142 "呼び出し SUB_001"
          SUB_001()
        elif (1401 == switch_1):
          $ 143 "ケース 1401"
          $ 144 "設定 GPIO_SubPrgNo=141"
          write_output_integer_register(2, 141)
          $ 145 "呼び出し SUB_141"
          SUB_141()
          $ 146 "pBucket[WorkPosNo]=Y2"
          pBucket[WorkPosNo]=Y2
          $ 147 "設定 GPIO_SubPrgNo=143"
          write_output_integer_register(2, 143)
          $ 148 "呼び出し SUB_143"
          SUB_143()
          $ 149 "設定 GPBO_BKPosDone=HI:Pulse 1.0"
          thread SinglePulse2259():
            write_output_boolean_register(13, True)
            sleep(1.0)
            write_output_boolean_register(13, False)
          end
          singlePulse2259 = run SinglePulse2259()
        elif (1402 == switch_1):
          $ 150 "ケース 1402"
          $ 151 "設定 GPIO_SubPrgNo=142"
          write_output_integer_register(2, 142)
          $ 152 "呼び出し SUB_142"
          SUB_142()
          $ 153 "設定 GPIO_SubPrgNo=001"
          write_output_integer_register(2, 001)
          $ 154 "呼び出し SUB_001"
          SUB_001()
          $ 155 "pCV=Y2"
          pCV=Y2
        elif (3100 == switch_1):
          $ 156 "ケース 3100"
          $ 157 "設定 GPIO_SubPrgNo=3100"
          write_output_integer_register(2, 3100)
          $ 158 "呼び出し SUB_3100"
          SUB_3100()
        elif (6001 == switch_1):
          $ 159 "ケース 6001"
          $ 160 "設定 GPIO_SubPrgNo=6001"
          write_output_integer_register(2, 6001)
          $ 161 "呼び出し SUB_6001"
          SUB_6001()
        elif (6101 == switch_1):
          $ 162 "ケース 6101"
          $ 163 "CheckMST:=0"
          global CheckMST=0
          $ 164 "設定 GPIO_SubPrgNo=6101"
          write_output_integer_register(2, 6101)
          $ 165 "呼び出し SUB_6101"
          SUB_6101()
        elif (6102 == switch_1):
          $ 166 "ケース 6102"
          $ 167 "If文 (GPII_CheckMST>0)"
          if ((read_input_integer_register(23)>0)):
            $ 168 "CheckMST:=GPII_CheckMST"
            global CheckMST=read_input_integer_register(23)
            $ 169 "WorkPosNo:=-1"
            global WorkPosNo=-1
            $ 170 "CaptRowNo:=5"
            global CaptRowNo=5
            $ 172 "SET_BUCKET()"
            SET_BUCKET()
            $ 173 "設定 GPIO_SubPrgNo=6101"
            write_output_integer_register(2, 6101)
            $ 174 "呼び出し SUB_6101"
            SUB_6101()
          end
          $ 175 "設定 GPIO_SubPrgNo=6102"
          write_output_integer_register(2, 6102)
          $ 179 "呼び出し SUB_6102RXFF"
          SUB_6102RXFF()
        elif (6401 == switch_1):
          $ 180 "ケース 6401"
          $ 181 "設定 GPIO_SubPrgNo=141"
          write_output_integer_register(2, 141)
          $ 182 "呼び出し SUB_141"
          SUB_141()
          $ 183 "pBucketM=Y2"
          pBucketM=Y2
          $ 184 "pBucket[WorkPosNo]=Y2"
          pBucket[WorkPosNo]=Y2
        elif (6402 == switch_1):
          $ 185 "ケース 6402"
          $ 186 "設定 GPIO_SubPrgNo=142"
          write_output_integer_register(2, 142)
          $ 187 "呼び出し SUB_6402"
          SUB_6402()
        elif (7001 == switch_1):
          $ 188 "ケース 7001"
          $ 189 "設定 GPIO_SubPrgNo=7001"
          write_output_integer_register(2, 7001)
          $ 190 "呼び出し SUB_7001"
          SUB_7001()
        elif (7002 == switch_1):
          $ 191 "ケース 7002"
          $ 192 "設定 GPIO_SubPrgNo=7002"
          write_output_integer_register(2, 7002)
          $ 193 "呼び出し SUB_7002"
          SUB_7002()
        end
        thread_flag_37 = 1
      end
      if ((SubPrgResult == 100)):
        global thread_handler_37=run Thread_if_37()
        while (thread_flag_37 == 0):
          if not((SubPrgResult == 100)):
            kill thread_handler_37
            thread_flag_37 = 2
          else:
            sync()
          end
        end
      else:
        thread_flag_37 = 2
      end
      $ 194 "設定 GPIO_PrgResult=SubPrgResult"
      write_output_integer_register(1, SubPrgResult)
      thread_flag_31 = 1
    end
    if ((  not  read_input_boolean_register(5) !=   False  )):
      global thread_handler_31=run Thread_if_31()
      while (thread_flag_31 == 0):
        if not((  not  read_input_boolean_register(5) !=   False  )):
          kill thread_handler_31
          thread_flag_31 = 2
        else:
          sync()
        end
      end
    else:
      thread_flag_31 = 2
    end
    $ 195 "END_CYCLE()"
    END_CYCLE()
    $ 196 "If文 GPBI_PrgStop≟ True "
    if (read_input_boolean_register(5) ==   True  ):
      $ 197 "SubPrgResult:=800"
      global SubPrgResult=800
      $ 198 "設定 GPIO_PrgResult=SubPrgResult"
      write_output_integer_register(1, SubPrgResult)
      $ 199 "設定 GPBO_PrgRun= False "
      write_output_boolean_register(6,   False  )
    end
    $ 200 "待機: 0.1"
    sleep(0.1)
    $ 201 "prg_no:=0"
    global prg_no=0
    $ 202 "荷重の設定: k10"
    set_target_payload(0.100000, [0.135000, 0.000000, 0.225000], [10.000000, 10.000000, 10.000000, 0.000000, 0.000000, 0.000000])
    $ 203 "設定"
    set_tcp(p[0.0,0.09,0.42,0.0,0.0,0.0])
    $ 204 "If文 (GPIO_PrgNo≠0)"
    if ((read_output_integer_register(0) != 0)):
      $ 205 "設定 GPBO_PrgEnd=HI:Pulse 1.0"
      thread SinglePulse2260():
        write_output_boolean_register(5, True)
        sleep(1.0)
        write_output_boolean_register(5, False)
      end
      singlePulse2260 = run SinglePulse2260()
      $ 206 "設定 GPIO_PrgNo=0"
      write_output_integer_register(0, 0)
    end
    $ 207 "待機 GPBI_PrgStart=LO"
    while (read_input_boolean_register(4) == True):
      sync()
    end
    $ 208 "待機 GPBI_PrgStop=LO"
    while (read_input_boolean_register(5) == True):
      sync()
    end
  end
end
